# B&R Automation Studio project CamAutomat1
Automation Studio 4.10.5.38 SP; technology packages: mapp 5.23.1, mappCockpit 5.23.0, mappControl 5.23.0, mappMotion 5.23.1, mappView 5.23.0

## Configuration Config1

CPU 5PPC2100.BY44-000, AutomationRuntime A4.83, Build 4.1.2, Safety 0.0, Vc 

CPU 5PPC2200.AL14-000, AutomationRuntime B4.91, Build 4.1.2, Safety 0.0, Vc 

### Task classes (Cpu.sw)
```
Cyclic#1 (cycle 2000 us, tolerance 2000 us):
  CamAutomat <- CamAutomat.prg
  SesnorSim <- SesnorSim.prg
Cyclic#3:
  ComTCP_P <- Libraries.ComTCP.ComTCP_P.prg
Cyclic#4:
  MachineAla <- MachineAlarm.prg
DataObjects: McAcpSys
NcDataObjects: McDriveLog
Binaries: TCData, mvLoader, TCLang, udbdef, arsvcreg, mCoWebSc, arflatprv, arcoal, McAcpDrv, McAcpSim, arconfig, asfw, ashwd, iomap, User, Role, sysconf, TC, ashwac, Config_2, Config, Config_1, Settings, Config_6, TempConfig, Config_7, Config_5, Config_3, Config_4
Libraries: MTBasics, brsystem, MTTypes, sys_lib, runtime, ComTCP_L, operator, astime, AsTCP, standard, AsArLog, AsBrStr, MpRecipe, MpBase, McBase, CoTrace, AsZip, FileIO, MpAxis, McAxis, McAcpAx, MpServer, MpAlarmX, MpCom, MpTemp, asieccon, arssl, asepl, powerlnk, aruser, dataobj
```

### Task classes (Cpu.sw)
```
Cyclic#1 (cycle 2000 us, tolerance 2000 us):
  CamAutomat <- CamAutomat.prg
  TouchProbe <- TouchProbe.prg
Cyclic#4:
  MachineAla <- MachineAlarm.prg
DataObjects: McAcpSys
NcDataObjects: McDriveLog
Binaries: TCData, mvLoader, TCLang, udbdef, arsvcreg, mCoWebSc, arflatprv, arcoal, McAcpDrv, McAcpSim, arconfig, asfw, ashwd, iomap, User, Role, sysconf, TC, ashwac, Config_2, Config, Config_1, Settings, Config_6, TempConfig, Config_5, CamAutom, Config_7, Config_3, Config_4
Libraries: MTBasics, brsystem, MTTypes, sys_lib, runtime, ComTCP_L, operator, astime, AsTCP, standard, AsArLog, AsBrStr, MpRecipe, MpBase, McBase, CoTrace, AsZip, FileIO, MpAxis, McAxis, McAcpAx, MpServer, MpAlarmX, MpCom, MpTemp, asieccon, arssl, asepl, powerlnk, aruser, dataobj
```

### Hardware
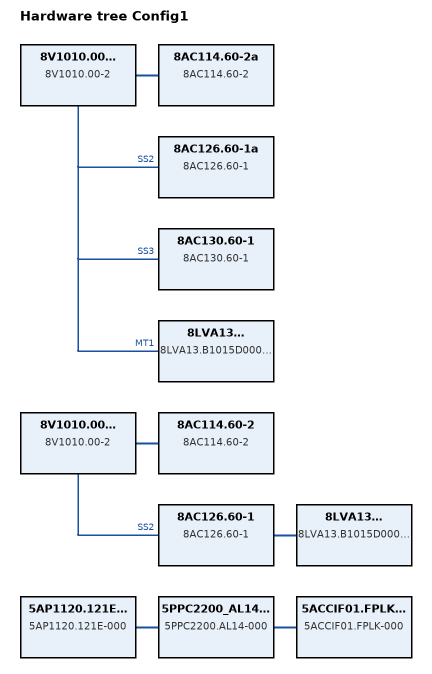
```
5ACCIF01.FPLK-000 : 5ACCIF01.FPLK-000 v1.6.2.0  [SL -> 5PPC2200_AL14_000.SL1]
5AP1120.121E-000 : 5AP1120.121E-000 v2.0.0.0
5PPC2200_AL14_000 : 5PPC2200.AL14-000 v2.0.1.0  [SY -> 5AP1120.121E-000.SY1]
  Connector IF3:
    AssignedOperatingSystem = ARemb
    ActivateDevice = 1
    HostName = mo
    Mode = Manual
    InternetAddress = 192.168.68.70
    SubnetMask = 255.255.255.0
    ActivateSnmp = 2
  Connector IF4:
    AssignedOperatingSystem = GPOS
  Connector IF7:
    OperatingSystem = ARemb
    ActivateDevice = 1
    Mode = Manual
    InternetAddress = 192.168.0.10
    SubnetMask = 255.255.255.0
  Connector IF5:
    AssignedOperatingSystem = ARemb
  Connector IF6:
    AssignedOperatingSystem = GPOS
  ConfigurationID = mappViewGettingStarted_ETA210_T50
  UserPartitionSize = 200
  RemMemDevice = PCI.1.PPC21xx.SRAM
  RemMemSize = 262144
  RemanentGlobalPvSize = 60000
  TimerDeviceType = EPLX2X
  TimerDevice = 5ACCIF01.FPLK-000.IF1
  TaskClassIdleTime = 2000
  Cyclic1Duration = 2000
  Cyclic1Tolerance = 2000
  FileDevice1
  FileDeviceName1 = CSV_Recipes
  FileDevicePath1 = F:\Recipes
  FileDevice2
  FileDeviceName2 = SIM_Recipes
  FileDevicePath2 = C:\Basic
  TimeZone = 65
  FtpUser1
  FtpUsername1 = academy
  FtpUserPassword1 = PTbbKbjlQWNQQLeLnvYxsprPr7USEpMWmZovrSfugvI=
  FtpUserSalt1 = LwThsYzd
  FTPAccessRight1 = 0
  ActivateOpcUa = 1
  OpcUa_SamplingTimer_Selector = 1
  OpcUaInformationModels_PV_Version = 1
  ActivateHypervisor = 1
8AC114.60-2 : 8AC114.60-2 v1.0.0.8  [SS -> 8V1010.00-2Cutter.SS1; PLK1 -> 8AC114.60-2a.PLK1 (NodeNumber=1) [Cable Type=PowerlinkCable, Length=10, Version=1.0.0.3]; PLK2 -> 5ACCIF01.FPLK-000.IF1 (NodeNumber=1) [Cable Type=PowerlinkCable, Length=10, Version=1.0.0.3]]
8AC114.60-2a : 8AC114.60-2 v1.0.0.8  [SS -> 8V1010.00-2aConv.SS1; PLK1 -> 8AC114.60-2.PLK1 (NodeNumber=2) [Cable Type=PowerlinkCable, Length=10, Version=1.0.0.3]]
8AC126.60-1 : 8AC126.60-1 v2.2.0.0  [SS -> 8V1010.00-2Cutter.SS2]
  PlugInType = Encoder
  McAcoposTypeID = AcoposPlugInConfig
8AC126.60-1a : 8AC126.60-1 v2.2.0.0  [SS -> 8V1010.00-2aConv.SS2]
  PlugInType = Encoder
  McAcoposTypeID = AcoposPlugInConfig
8AC130.60-1 : 8AC130.60-1 v2.2.0.0  [SS -> 8V1010.00-2aConv.SS3]
8LVA13.B1015D000-0 : 8LVA13.B1015D000-0 v2.2.0.3  [EC -> 8AC126.60-1.EC; MT -> 8V1010.00-2Cutter.MT1]
  M1/MotorParameters:
    MOTOR_AMB_TEMP_RATED = 40
8LVA13.B1015D000-0a : 8LVA13.B1015D000-0 v2.2.0.3  [MT -> 8V1010.00-2aConv.MT1]
  M1/MotorParameters:
    MOTOR_AMB_TEMP_RATED = 40
8V1010.00-2Cutter : 8V1010.00-2 v2.3.0.0  // Cutter ACOPOS servo drive, 3x 400-480 V, 1.0 A, 0.45 kW, line filter, integrated braking resistor and electronic secure restart inhibit
  DriveConfiguration/Module:
    McAcoposTypeID = AcoposConfig
    ActivateACOPOSSimulationOnPLC = 0
    PowerSupply = ETA
  DriveConfiguration/Channel[1]/RealAxis:
    AxisReference = gCutter_MpLink
    MechanicalElementsIsInvisible = 0
  DriveConfiguration/Channel[1]/RealAxis/MechanicalElements/Gearbox:
    InputIsReadOnly = 0
    Input = 1
    OutputIsReadOnly = 0
    Output = 1
  DriveConfiguration/Channel[1]/RealAxis/MechanicalElements/RotaryToLinearTransformation:
    ReferenceDistanceIsReadOnly = 0
    ReferenceDistance = 360
  DriveConfiguration/Channel[1]/RealAxis/Controller:
    ModeIsReadOnly = 0
    Mode = PositionController
  DriveConfiguration/Channel[1]/RealAxis/Controller/Mode/Position:
    ProportionalGain = 228
    IntegrationTime = 0.0
    PredictionTime = 0.0004
    TotalDelayTime = 0.0004
  DriveConfiguration/Channel[1]/RealAxis/Controller/Mode/Speed:
    ProportionalGainIsReadOnly = 0
    ProportionalGain = 0.599999
    IntegrationTimeIsReadOnly = 0
    IntegrationTime = 0.0
    FilterTimeIsReadOnly = 0
    FilterTime = 0.0
  DriveConfiguration/Channel[1]/RealAxis/Controller/Mode/LoopFilters:
    LoopFilterXIsReadOnly = 0
    LoopFilter1 = NotUsed
    LoopFilter2 = NotUsed
    LoopFilter3 = NotUsed
  DriveConfiguration/Channel[1]/RealAxis/Homing:
    ModeIsReadOnly = 0
    Mode = Direct
  DriveConfiguration/Channel[1]/RealAxis/Homing/Mode:
    Position = 0.0
    ReferencePulse = NotUsed
  DriveConfiguration/Channel[1]/RealAxis/Homing:
    RestorePositionVariable = 
  DriveConfiguration/Channel[1]/RealAxis/StopReaction:
    QuickstopIsReadOnly = 0
    Quickstop = DecelerationLimit
    DriveErrorIsReadOnly = 0
    DriveError = DecelerationLimit
  DriveConfiguration/Channel[1]/RealAxis/MovementErrorLimits:
    PositionError = 1
    VelocityErrorMonitoring = Automatic1
  DriveConfiguration/Channel[1]/RealAxis:
    JerkFilterIsReadOnly = 0
    JerkFilter = NotUsed
    ZeroVibrationFilter = NotUsed
  DriveConfiguration/Channel[1]/RealAxis/DigitalInputs/HomingSwitch:
    SourceIsReadOnly = 0
    Source = X1Ref
    Level = High
  DriveConfiguration/Channel[1]/RealAxis/DigitalInputs/PositiveLimitSwitch:
    Source = X1PosLim
    Level = High
  DriveConfiguration/Channel[1]/RealAxis/DigitalInputs/NegativeLimitSwitch:
    Source = X1NegLim
    Level = High
  DriveConfiguration/Channel[1]/RealAxis/DigitalInputs/Trigger1:
    Source = X1Trigger1
    Level = High
  DriveConfiguration/Channel[1]/RealAxis/DigitalInputs/Trigger2:
    Source = X1Trigger2
    Level = High
  DriveConfiguration/Channel[1]/RealAxis/DigitalInputs/Quickstop:
    Input = NotUsed
  DriveConfiguration/Channel[1]/RealAxis/Simulation:
    SimulationModeOnPLC = SetValueGeneration
    SimulationModeOnACOPOS = NotUsed
  DriveConfiguration/Channel[1]/RealAxis/AxisFeatures:
    FeatureRef[1] = Feature_CamAutomat
  DriveConfiguration/Channel[1]:
    ExternalEncoderAxis = NotUsed
8V1010.00-2aConv : 8V1010.00-2 v2.3.0.0  // Conv ACOPOS servo drive, 3x 400-480 V, 1.0 A, 0.45 kW, line filter, integrated braking resistor and electronic secure restart inhibit
  DriveConfiguration/Module:
    McAcoposTypeID = AcoposConfig
    ActivateACOPOSSimulationOnPLC = 0
    PowerSupply = ETA
  DriveConfiguration/Channel[1]/RealAxis:
    AxisReference = gConv_MpLink
    MechanicalElementsIsInvisible = 0
  DriveConfiguration/Channel[1]/RealAxis/MechanicalElements/Gearbox:
    InputIsReadOnly = 0
    Input = 1
    OutputIsReadOnly = 0
    Output = 1
  DriveConfiguration/Channel[1]/RealAxis/MechanicalElements/RotaryToLinearTransformation:
    ReferenceDistanceIsReadOnly = 0
    ReferenceDistance = 160
  DriveConfiguration/Channel[1]/RealAxis/Controller:
    ModeIsReadOnly = 0
    Mode = PositionController
  DriveConfiguration/Channel[1]/RealAxis/Controller/Mode/Position:
    ProportionalGain = 269
    IntegrationTime = 0.0
    PredictionTime = 0.0004
    TotalDelayTime = 0.0004
  DriveConfiguration/Channel[1]/RealAxis/Controller/Mode/Speed:
    ProportionalGainIsReadOnly = 0
    ProportionalGain = 0.45
    IntegrationTimeIsReadOnly = 0
    IntegrationTime = 0.0
    FilterTimeIsReadOnly = 0
    FilterTime = 0.0
  DriveConfiguration/Channel[1]/RealAxis/Controller/Mode/LoopFilters:
    LoopFilterXIsReadOnly = 0
    LoopFilter1 = NotUsed
    LoopFilter2 = NotUsed
    LoopFilter3 = NotUsed
  DriveConfiguration/Channel[1]/RealAxis/Homing:
    ModeIsReadOnly = 0
    Mode = Direct
  DriveConfiguration/Channel[1]/RealAxis/Homing/Mode:
    Position = 0.0
    ReferencePulse = NotUsed
  DriveConfiguration/Channel[1]/RealAxis/Homing:
    RestorePositionVariable = 
  DriveConfiguration/Channel[1]/RealAxis/StopReaction:
    QuickstopIsReadOnly = 0
    Quickstop = DecelerationLimit
    DriveErrorIsReadOnly = 0
    DriveError = DecelerationLimit
  DriveConfiguration/Channel[1]/RealAxis/MovementErrorLimits:
    PositionError = 1
    VelocityErrorMonitoring = Automatic1
  DriveConfiguration/Channel[1]/RealAxis:
    JerkFilterIsReadOnly = 0
    JerkFilter = NotUsed
    ZeroVibrationFilter = NotUsed
  DriveConfiguration/Channel[1]/RealAxis/DigitalInputs/HomingSwitch:
    SourceIsReadOnly = 0
    Source = X1Ref
    Level = High
  DriveConfiguration/Channel[1]/RealAxis/DigitalInputs/PositiveLimitSwitch:
    Source = X1PosLim
    Level = High
  DriveConfiguration/Channel[1]/RealAxis/DigitalInputs/NegativeLimitSwitch:
    Source = X1NegLim
    Level = High
  DriveConfiguration/Channel[1]/RealAxis/DigitalInputs/Trigger1:
    Source = X1Trigger1
    Level = High
  DriveConfiguration/Channel[1]/RealAxis/DigitalInputs/Trigger2:
    Source = X1Trigger2
    Level = High
  DriveConfiguration/Channel[1]/RealAxis/DigitalInputs/Quickstop:
    Input = NotUsed
  DriveConfiguration/Channel[1]/RealAxis/Simulation:
    SimulationModeOnPLC = SetValueGeneration
    SimulationModeOnACOPOS = NotUsed
  DriveConfiguration/Channel[1]/RealAxis/AxisFeatures:
    FeatureRef[1] = 
  DriveConfiguration/Channel[1]:
    ExternalEncoderAxis = NotUsed
```

### TempConfig.tempcontroller - 5PPC2100_BY44_000/mappControl/TempConfig.tempcontroller
```
Element gTempController_2 (Type=tempcontroller)
  TempController:
    SoftStart = NotUsed
Element gTempController_1 (Type=tempcontroller)
  TempController:
    SoftStart = NotUsed
```

### CamAutom.axisfeature - 5PPC2100_BY44_000/mappMotion/CamAutom.axisfeature
```
Element Feature_CamAutomat_1 (Type=axisfeature)
  Type = CamAutomat
    CamAutomatType = ACOPOS
      CommonParameters:
        Master:
          ValueSource = SetPosition
            AxisReference = gAxis1_MpLink
            MaxVelocity = 1000
          StartPosition = 0.0
          StartInterval = MasterAxisPeriod
        AdvancedParameters:
          StartStateParameters:
            StartState = 0
            RelMasterStartPos = 0.0
          AdditiveAxes:
            AdditiveMasterValueSource = NotUsed
            AdditiveSlaveValueSource = NotUsed
          MasterStartPositionMode = NotEvaluatedAnew
          ControlSettings:
            CrossLeftBoundary = PositionLimitedHorizontal
            CamChangeImmediately = CurrentMasterMoveDir
          MessageSettings:
            ErrorsInStandby = NoErrorMessages
          TriggerAndLatch:
            Trigger1Delay = 0.0
            Trigger2Delay = 0.0
            SlaveLatchParID = 0
          EventParIDs
          StartIntervals
          Factors:
            SlaveFactorParID = 0
      States:
        State0 = Used
          Events:
            Event[0]:
              Type = MasterStartPosition
              Transition = Immediately
              SynchronousUpdate = NotUsed
              NextState = 1
        State[1]:
          Cam = Predefined
            PredefinedCam = OneToOne
          MasterFactor = 72
          SlaveFactor = 0
          CompensationMode = DistancesBetweenCamCenterPoints
            MasterDistance = 288
            SlaveDistance = 0.0
            AdvancedParameters = NotUsed
          AdvancedParameters:
            RepeatCounterInit = 0
            MasterValueSource = CommonMaster
          Events:
            Event[0]:
              Type = Signal1FromPLC
              Transition = EndOfState
              SynchronousUpdate = NotUsed
              NextState = 2
        State[2]:
          Cam = Predefined
            PredefinedCam = OneToOne
          MasterFactor = 72
          SlaveFactor = 72
          CompensationMode = MaDistBetweenLatchPosCenter
            MasterDistance = 144
            SlaveDistance = 144
            AdvancedParameters = NotUsed
          AdvancedParameters:
            RepeatCounterInit = 0
            MasterValueSource = CommonMaster
          Events:
            Event[0]:
              Type = Signal1FromPLC
              Transition = EndOfState
              SynchronousUpdate = NotUsed
              NextState = 3
            Event[1]:
              Type = StateEnd
              Transition = EndOfState
              SynchronousUpdate = NotUsed
              NextState = 4
        State[3]:
          Cam = Predefined
            PredefinedCam = OneToOne
          MasterFactor = 72
          SlaveFactor = 72
          CompensationMode = MaDistBetweenLatchPosCenter
            MasterDistance = 288
            SlaveDistance = 288
            AdvancedParameters = NotUsed
          AdvancedParameters:
            RepeatCounterInit = 0
            MasterValueSource = CommonMaster
          Events:
            Event[0]:
              Type = Signal1FromPLC
              Transition = EndOfState
              SynchronousUpdate = NotUsed
              NextState = 3
            Event[1]:
              Type = StateEnd
              Transition = EndOfState
              SynchronousUpdate = NotUsed
              NextState = 4
        State[4]:
          Cam = Predefined
            PredefinedCam = OneToOne
          MasterFactor = 72
          SlaveFactor = 0
          CompensationMode = MaDistBetweenLatchPosCenter
            MasterDistance = 144
            SlaveDistance = 144
            AdvancedParameters = NotUsed
          AdvancedParameters:
            RepeatCounterInit = 0
            MasterValueSource = CommonMaster
          Events:
            Event[0]:
              Type = Signal1FromPLC
              Transition = EndOfState
              SynchronousUpdate = NotUsed
              NextState = 2
            Event[1]:
              Type = StateEnd
              Transition = EndOfState
              SynchronousUpdate = NotUsed
              NextState = 1
Element Feature_CamAutomat (Type=axisfeature)
  Type = CamAutomat
    CamAutomatType = ACOPOS
      CommonParameters:
        Master:
          ValueSource = SetPosition
            AxisReference = gAxis1_MpLink
            MaxVelocity = 1000
          StartPosition = 0.0
          StartInterval = MasterAxisPeriod
        AdvancedParameters:
          StartStateParameters:
            StartState = 0
            RelMasterStartPos = 0.0
          AdditiveAxes:
            AdditiveMasterValueSource = NotUsed
            AdditiveSlaveValueSource = NotUsed
          MasterStartPositionMode = NotEvaluatedAnew
          ControlSettings:
            CrossLeftBoundary = PositionLimitedHorizontal
            CamChangeImmediately = CurrentMasterMoveDir
          MessageSettings:
            ErrorsInStandby = NoErrorMessages
          TriggerAndLatch:
            Trigger1Delay = 0.0
            Trigger2Delay = 0.0
            SlaveLatchParID = 0
          EventParIDs
          StartIntervals
          Factors:
            SlaveFactorParID = 0
      States:
        State0 = Used
          Events:
            Event[0]:
              Type = MasterStartPosition
              Transition = Immediately
              SynchronousUpdate = NotUsed
              NextState = 1
        State[1]:
          Cam = Predefined
            PredefinedCam = OneToOne
          MasterFactor = 1
          SlaveFactor = 0
          CompensationMode = DistancesBetweenCamCenterPoints
            MasterDistance = 0.0
            SlaveDistance = 0.0
            AdvancedParameters = NotUsed
          AdvancedParameters:
            RepeatCounterInit = 0
            MasterValueSource = CommonMaster
          Events:
            Event[0]:
              Type = Signal1FromPLC
              Transition = EndOfState
              SynchronousUpdate = NotUsed
              NextState = 2
        State[2]:
          Cam = Predefined
            PredefinedCam = OneToOne
          MasterFactor = 1
          SlaveFactor = 1
          CompensationMode = MaDistBetweenLatchPosCenter
            MasterDistance = 130
            SlaveDistance = 170
            AdvancedParameters = NotUsed
          AdvancedParameters:
            RepeatCounterInit = 0
            MasterValueSource = CommonMaster
          Events:
            Event[0]:
              Type = StateEnd
              Transition = EndOfState
              SynchronousUpdate = NotUsed
              NextState = 3
        State[3]:
          Cam = Predefined
            PredefinedCam = OneToOne
          MasterFactor = 1
          SlaveFactor = 1
          CompensationMode = MaDistBetweenLatchPosCenter
            MasterDistance = 20
            SlaveDistance = 20
            AdvancedParameters = NotUsed
          AdvancedParameters:
            RepeatCounterInit = 0
            MasterValueSource = CommonMaster
          Events:
            Event[0]:
              Type = StateEnd
              Transition = EndOfState
              SynchronousUpdate = NotUsed
              NextState = 4
        State[4]:
          Cam = Predefined
            PredefinedCam = OneToOne
          MasterFactor = 1
          SlaveFactor = 0
          CompensationMode = MaDistBetweenLatchPosCenter
            MasterDistance = 130
            SlaveDistance = 170
            AdvancedParameters = NotUsed
          AdvancedParameters:
            RepeatCounterInit = 0
            MasterValueSource = CommonMaster
          Events:
            Event[0]:
              Type = StateEnd
              Transition = EndOfState
              SynchronousUpdate = NotUsed
              NextState = 1
```

### Config_1.axis - 5PPC2100_BY44_000/mappMotion/Config_1.axis
```
Element gAxis2_MpLink (Type=axis)
  BaseTypeIsReadOnly = 0
  BaseType = RotaryPeriodic
    MeasurementUnitIsReadOnly = 0
    MeasurementUnit = 17476
    MeasurementResolutionIsReadOnly = 0
    MeasurementResolution = 1
    CountDirectionIsReadOnly = 0
    CountDirection = Standard
    PeriodSettings:
      Period = 360.0
  MovementLimitsIsReadOnly = 0
  MovementLimits = Internal
    Position:
      LowerLimitMin = -1.79769313486231E308
      UpperLimitMax = 1.79769313486231E308
      LowerLimit = -1000.0
      UpperLimit = 1000.0
    VelocityIsReadOnly = 0
    Velocity:
      VelocityMax = 3.4E38
      Velocity = 6000
    AccelerationIsReadOnly = 0
    Acceleration:
      AccelerationMax = 3.4E38
      Acceleration = 60000
    DecelerationIsReadOnly = 0
    Deceleration:
      DecelerationMax = 3.4E38
      Deceleration = 60000
  Alarms = MpAlarmX
Element gAxis1_MpLink (Type=axis)
  BaseTypeIsReadOnly = 0
  BaseType = RotaryPeriodic
    MeasurementUnitIsReadOnly = 0
    MeasurementUnit = 17476
    MeasurementResolutionIsReadOnly = 0
    MeasurementResolution = 1
    CountDirectionIsReadOnly = 0
    CountDirection = Standard
    PeriodSettings:
      Period = 360.0
  MovementLimitsIsReadOnly = 0
  MovementLimits = Internal
    Position:
      LowerLimitMin = -1.79769313486231E308
      UpperLimitMax = 1.79769313486231E308
      LowerLimit = -1000.0
      UpperLimit = 1000.0
    VelocityIsReadOnly = 0
    Velocity:
      VelocityMax = 3.4E38
      Velocity = 6000
    AccelerationIsReadOnly = 0
    Acceleration:
      AccelerationMax = 3.4E38
      Acceleration = 60000
    DecelerationIsReadOnly = 0
    Deceleration:
      DecelerationMax = 3.4E38
      Deceleration = 60000
  Alarms = MpAlarmX
```

### Axis.axis - 5PPC2200_AL14_000/mappMotion/Axis.axis
```
Element gConv_MpLink (Type=axis)  // Conver Servo
  BaseTypeIsReadOnly = 0
  BaseType = LinearPeriodic
    MeasurementUnit = 5066068
    MeasurementResolutionIsReadOnly = 0
    MeasurementResolution = 0.01
    CountDirectionIsReadOnly = 0
    CountDirection = Standard
    PeriodSettings:
      Period = 144
  MovementLimitsIsReadOnly = 0
  MovementLimits = Internal
    Position:
      LowerLimitMin = -1.79769313486231E308
      UpperLimitMax = 1.79769313486231E308
      LowerLimit = -1000.0
      UpperLimit = 1000.0
    VelocityIsReadOnly = 0
    Velocity:
      VelocityMax = 3.4E38
      Velocity = 6000
    AccelerationIsReadOnly = 0
    Acceleration:
      AccelerationMax = 3.4E38
      Acceleration = 60000
    DecelerationIsReadOnly = 0
    Deceleration:
      DecelerationMax = 3.4E38
      Deceleration = 60000
  Alarms = MpAlarmX
Element gCutter_MpLink (Type=axis)  // Cutter Servo
  BaseTypeIsReadOnly = 0
  BaseType = RotaryPeriodic
    MeasurementUnitIsReadOnly = 0
    MeasurementUnit = 17476
    MeasurementResolutionIsReadOnly = 0
    MeasurementResolution = 0.01
    CountDirectionIsReadOnly = 0
    CountDirection = Inverse
    PeriodSettings:
      Period = 360
  MovementLimitsIsReadOnly = 0
  MovementLimits = Internal
    Position:
      LowerLimitMin = -1.79769313486231E308
      UpperLimitMax = 1.79769313486231E308
      LowerLimit = -1000.0
      UpperLimit = 1000.0
    VelocityIsReadOnly = 0
    Velocity:
      VelocityMax = 3.4E38
      Velocity = 6000
    AccelerationIsReadOnly = 0
    Acceleration:
      AccelerationMax = 3.4E38
      Acceleration = 60000
    DecelerationIsReadOnly = 0
    Deceleration:
      DecelerationMax = 3.4E38
      Deceleration = 60000
  Alarms = MpAlarmX
```

### CamAutom.axisfeature - 5PPC2200_AL14_000/mappMotion/CamAutom.axisfeature
```
Element Feature_CamAutomatbak (Type=axisfeature)
  Type = CamAutomat
    CamAutomatType = ACOPOS
      CommonParameters:
        Master:
          ValueSource = SetPosition
            AxisReference = gConv_MpLink
            MaxVelocity = 1000
          StartPosition = 0.00
          StartInterval = MasterAxisPeriod
        AdvancedParameters:
          StartStateParameters:
            StartState = 0
            RelMasterStartPos = 0.0
          AdditiveAxes:
            AdditiveMasterValueSource = NotUsed
            AdditiveSlaveValueSource = NotUsed
          MasterStartPositionMode = NotEvaluatedAnew
          ControlSettings:
            CrossLeftBoundary = PositionLimitedHorizontal
            CamChangeImmediately = CurrentMasterMoveDir
          MessageSettings:
            ErrorsInStandby = NoErrorMessages
          TriggerAndLatch:
            Trigger1Delay = 0.0
            Trigger2Delay = 0.0
            SlaveLatchParID = 0
          EventParIDs
          StartIntervals
          Factors:
            SlaveFactorParID = 0
      States:
        State0 = Used
          Events:
            Event[0]:
              Type = MasterStartPosition
              Transition = Immediately
              SynchronousUpdate = NotUsed
              NextState = 1
        State[1]:
          Cam = Predefined
            PredefinedCam = OneToOne
          MasterFactor = 100
          SlaveFactor = 0
          CompensationMode = DistancesBetweenExitEntryPoints
            MasterDistance = 0
            SlaveDistance = 0
            AdvancedParameters = NotUsed
          AdvancedParameters:
            RepeatCounterInit = 0
            MasterValueSource = CommonMaster
          Events:
            Event[0]:
              Type = Signal1FromPLC
              Transition = EndOfState
              SynchronousUpdate = NotUsed
              NextState = 2
        State[2]:
          Cam = Predefined
            PredefinedCam = OneToOne
          MasterFactor = 2000
          SlaveFactor = 2300
          CompensationMode = DistancesBetweenExitEntryPoints
            MasterDistance = 100
            SlaveDistance = 160
            AdvancedParameters = NotUsed
          AdvancedParameters:
            RepeatCounterInit = 0
            MasterValueSource = CommonMaster
          Events:
            Event[0]:
              Type = StateEnd
              Transition = EndOfState
              SynchronousUpdate = NotUsed
              NextState = 3
        State[3]:
          Cam = Predefined
            PredefinedCam = OneToOne
          MasterFactor = 100
          SlaveFactor = 0
          CompensationMode = DistancesBetweenExitEntryPoints
            MasterDistance = 1
            SlaveDistance = 288
            AdvancedParameters = NotUsed
          AdvancedParameters:
            RepeatCounterInit = 0
            MasterValueSource = CommonMaster
          Events:
            Event[0]:
              Type = Signal1FromPLC
              Transition = EndOfState
              SynchronousUpdate = NotUsed
              NextState = 3
            Event[1]:
              Type = StateEnd
              Transition = Immediately
              SynchronousUpdate = NotUsed
              NextState = 4
        State[4]:
          Cam = Predefined
            PredefinedCam = OneToOne
          MasterFactor = 72
          SlaveFactor = 0
          CompensationMode = DistancesBetweenExitEntryPoints
            MasterDistance = 144
            SlaveDistance = 144
            AdvancedParameters = NotUsed
          AdvancedParameters:
            RepeatCounterInit = 0
            MasterValueSource = CommonMaster
          Events:
            Event[0]:
              Type = Signal1FromPLC
              Transition = EndOfState
              SynchronousUpdate = NotUsed
              NextState = 2
            Event[1]:
              Type = StateEnd
              Transition = Immediately
              SynchronousUpdate = NotUsed
              NextState = 1
Element Feature_CamAutomat_3rd (Type=axisfeature)
  Type = CamAutomat
    CamAutomatType = ACOPOS
      CommonParameters:
        Master:
          ValueSource = SetPosition
            AxisReference = gConv_MpLink
            MaxVelocity = 1000
          StartPosition = 0.00
          StartInterval = MasterAxisPeriod
        AdvancedParameters:
          StartStateParameters:
            StartState = 0
            RelMasterStartPos = 0.0
          AdditiveAxes:
            AdditiveMasterValueSource = NotUsed
            AdditiveSlaveValueSource = NotUsed
          MasterStartPositionMode = NotEvaluatedAnew
          ControlSettings:
            CrossLeftBoundary = PositionLimitedHorizontal
            CamChangeImmediately = CurrentMasterMoveDir
          MessageSettings:
            ErrorsInStandby = NoErrorMessages
          TriggerAndLatch:
            Trigger1Delay = 0.0
            Trigger2Delay = 0.0
            SlaveLatchParID = 0
          EventParIDs
          StartIntervals
          Factors:
            SlaveFactorParID = 0
      States:
        State0 = Used
          Events:
            Event[0]:
              Type = MasterStartPosition
              Transition = Immediately
              SynchronousUpdate = NotUsed
              NextState = 1
        State[1]:
          Cam = Predefined
            PredefinedCam = OneToOne
          MasterFactor = 100
          SlaveFactor = 0
          CompensationMode = NoCompensation
          AdvancedParameters:
            RepeatCounterInit = 0
            MasterValueSource = CommonMaster
          Events:
            Event[0]:
              Type = Signal1FromPLC
              Transition = EndOfState
              SynchronousUpdate = NotUsed
              NextState = 2
        State[2]:
          Cam = Predefined
            PredefinedCam = OneToOne
          MasterFactor = 2000
          SlaveFactor = 2000
          CompensationMode = DistancesBetweenExitEntryPoints
            MasterDistance = 95
            SlaveDistance = 80
            AdvancedParameters = NotUsed
          AdvancedParameters:
            RepeatCounterInit = 0
            MasterValueSource = CommonMaster
          Events:
            Event[0]:
              Type = Signal1FromPLC
              Transition = EndOfState
              SynchronousUpdate = NotUsed
              NextState = 4
            Event[1]:
              Type = StateEnd
              Transition = EndOfState
              SynchronousUpdate = NotUsed
              NextState = 3
        State[3]:
          Cam = Predefined
            PredefinedCam = OneToOne
          MasterFactor = 100
          SlaveFactor = 0
          CompensationMode = NoCompensation
          AdvancedParameters:
            RepeatCounterInit = 0
            MasterValueSource = CommonMaster
          Events:
            Event[0]:
              Type = Signal1FromPLC
              Transition = EndOfState
              SynchronousUpdate = NotUsed
              NextState = 4
            Event[1]:
              Type = Signal2FromPLC
              Transition = Immediately
              SynchronousUpdate = NotUsed
              NextState = 5
        State[4]:
          Cam = Predefined
            PredefinedCam = OneToOne
          MasterFactor = 2000
          SlaveFactor = 2000
          CompensationMode = DistancesBetweenExitEntryPoints
            MasterDistance = 50
            SlaveDistance = 340
            AdvancedParameters = NotUsed
          AdvancedParameters:
            RepeatCounterInit = 0
            MasterValueSource = CommonMaster
          Events:
            Event[0]:
              Type = StateEnd
              Transition = Immediately
              SynchronousUpdate = NotUsed
              NextState = 3
        State[5]:
          Cam = Predefined
            PredefinedCam = OneToOne
          MasterFactor = 100
          SlaveFactor = 0
          CompensationMode = DistancesBetweenExitEntryPoints
            MasterDistance = 260
            SlaveDistance = 260
            AdvancedParameters = NotUsed
          AdvancedParameters:
            RepeatCounterInit = 0
            MasterValueSource = CommonMaster
          Events:
            Event[0]:
              Type = StateEnd
              Transition = EndOfState
              SynchronousUpdate = NotUsed
              NextState = 6
        State[6]:
          Cam = Predefined
            PredefinedCam = OneToOne
          MasterFactor = 100
          SlaveFactor = 0
          CompensationMode = NoCompensation
          AdvancedParameters:
            RepeatCounterInit = 0
            MasterValueSource = CommonMaster
Element Feature_CamAutomat_2nd (Type=axisfeature)
  Type = CamAutomat
    CamAutomatType = ACOPOS
      CommonParameters:
        Master:
          ValueSource = SetPosition
            AxisReference = gConv_MpLink
            MaxVelocity = 1000
          StartPosition = 0.00
          StartInterval = MasterAxisPeriod
        AdvancedParameters:
          StartStateParameters:
            StartState = 0
            RelMasterStartPos = 0.0
          AdditiveAxes:
            AdditiveMasterValueSource = NotUsed
            AdditiveSlaveValueSource = NotUsed
          MasterStartPositionMode = NotEvaluatedAnew
          ControlSettings:
            CrossLeftBoundary = PositionLimitedHorizontal
            CamChangeImmediately = CurrentMasterMoveDir
          MessageSettings:
            ErrorsInStandby = NoErrorMessages
          TriggerAndLatch:
            Trigger1Delay = 0.0
            Trigger2Delay = 0.0
            SlaveLatchParID = 0
          EventParIDs
          StartIntervals
          Factors:
            SlaveFactorParID = 0
      States:
        State0 = Used
          Events:
            Event[0]:
              Type = MasterStartPosition
              Transition = Immediately
              SynchronousUpdate = NotUsed
              NextState = 1
        State[1]:
          Cam = Predefined
            PredefinedCam = OneToOne
          MasterFactor = 100
          SlaveFactor = 0
          CompensationMode = NoCompensation
          AdvancedParameters:
            RepeatCounterInit = 0
            MasterValueSource = CommonMaster
          Events:
            Event[0]:
              Type = Signal1FromPLC
              Transition = EndOfState
              SynchronousUpdate = NotUsed
              NextState = 2
        State[2]:
          Cam = Predefined
            PredefinedCam = OneToOne
          MasterFactor = 2000
          SlaveFactor = 2000
          CompensationMode = DistancesBetweenExitEntryPoints
            MasterDistance = 95
            SlaveDistance = 160
            AdvancedParameters = NotUsed
          AdvancedParameters:
            RepeatCounterInit = 0
            MasterValueSource = CommonMaster
          Events:
            Event[0]:
              Type = Signal1FromPLC
              Transition = EndOfState
              SynchronousUpdate = NotUsed
              NextState = 4
            Event[1]:
              Type = StateEnd
              Transition = EndOfState
              SynchronousUpdate = NotUsed
              NextState = 3
        State[3]:
          Cam = Predefined
            PredefinedCam = OneToOne
          MasterFactor = 1000
          SlaveFactor = 1000
          CompensationMode = DistancesBetweenExitEntryPoints
            MasterDistance = 20
            SlaveDistance = 170
            AdvancedParameters = NotUsed
          AdvancedParameters:
            RepeatCounterInit = 0
            MasterValueSource = CommonMaster
          Events:
            Event[0]:
              Type = Signal1FromPLC
              Transition = EndOfState
              SynchronousUpdate = NotUsed
              NextState = 6
        State[4]:
          Cam = Predefined
            PredefinedCam = OneToOne
          MasterFactor = 2000
          SlaveFactor = 2000
          CompensationMode = DistancesBetweenExitEntryPoints
            MasterDistance = 95
            SlaveDistance = 340
            AdvancedParameters = NotUsed
          AdvancedParameters:
            RepeatCounterInit = 0
            MasterValueSource = CommonMaster
          Events:
            Event[0]:
              Type = Signal1FromPLC
              Transition = EndOfState
              SynchronousUpdate = NotUsed
              NextState = 5
            Event[1]:
              Type = StateEnd
              Transition = Immediately
              SynchronousUpdate = NotUsed
              NextState = 3
        State[5]:
          Cam = Predefined
            PredefinedCam = OneToOne
          MasterFactor = 2000
          SlaveFactor = 2000
          CompensationMode = DistancesBetweenExitEntryPoints
            MasterDistance = 95
            SlaveDistance = 340
            AdvancedParameters = NotUsed
          AdvancedParameters:
            RepeatCounterInit = 0
            MasterValueSource = CommonMaster
          Events:
            Event[0]:
              Type = Signal1FromPLC
              Transition = EndOfState
              SynchronousUpdate = NotUsed
              NextState = 4
            Event[1]:
              Type = StateEnd
              Transition = EndOfState
              SynchronousUpdate = NotUsed
              NextState = 3
        State[6]:
          Cam = Predefined
            PredefinedCam = OneToOne
          MasterFactor = 2000
          SlaveFactor = 2000
          CompensationMode = DistancesBetweenExitEntryPoints
            MasterDistance = 25
            SlaveDistance = 160
            AdvancedParameters = NotUsed
          AdvancedParameters:
            RepeatCounterInit = 0
            MasterValueSource = CommonMaster
          Events:
            Event[0]:
              Type = Signal1FromPLC
              Transition = EndOfState
              SynchronousUpdate = NotUsed
              NextState = 5
            Event[1]:
              Type = StateEnd
              Transition = EndOfState
              SynchronousUpdate = NotUsed
              NextState = 3
Element Feature_CamAutomat_finalok (Type=axisfeature)
  Type = CamAutomat
    CamAutomatType = ACOPOS
      CommonParameters:
        Master:
          ValueSource = SetPosition
            AxisReference = gConv_MpLink
            MaxVelocity = 1000
          StartPosition = 0.00
          StartInterval = SpecifyValue
            Interval = 1.0
        AdvancedParameters:
          StartStateParameters:
            StartState = 0
            RelMasterStartPos = 0.0
          AdditiveAxes:
            AdditiveMasterValueSource = NotUsed
            AdditiveSlaveValueSource = NotUsed
          MasterStartPositionMode = NotEvaluatedAnew
          ControlSettings:
            CrossLeftBoundary = PositionLimitedHorizontal
            CamChangeImmediately = CurrentMasterMoveDir
          MessageSettings:
            ErrorsInStandby = NoErrorMessages
          TriggerAndLatch:
            Trigger1Delay = 0.0
            Trigger2Delay = 0.0
            SlaveLatchParID = 0
          EventParIDs
          StartIntervals
          Factors:
            SlaveFactorParID = 0
      States:
        State0 = Used
          Events:
            Event[0]:
              Type = MasterStartPosition
              Transition = Immediately
              SynchronousUpdate = NotUsed
              NextState = 1
        State[1]:
          Cam = Predefined
            PredefinedCam = OneToOne
          MasterFactor = 100
          SlaveFactor = 0
          CompensationMode = NoCompensation
          AdvancedParameters:
            RepeatCounterInit = 0
            MasterValueSource = CommonMaster
          Events:
            Event[0]:
              Type = Signal1FromPLC
              Transition = EndOfState
              SynchronousUpdate = NotUsed
              NextState = 2
        State[2]:
          Cam = Predefined
            PredefinedCam = OneToOne
          MasterFactor = 100
          SlaveFactor = 0
          CompensationMode = DistancesBetweenExitEntryPoints
            MasterDistance = 27
            SlaveDistance = 80
            AdvancedParameters = NotUsed
          AdvancedParameters:
            RepeatCounterInit = 0
            MasterValueSource = CommonMaster
          Events:
            Event[0]:
              Type = StateEnd
              Transition = EndOfState
              SynchronousUpdate = NotUsed
              NextState = 3
        State[3]:
          Cam = Predefined
            PredefinedCam = OneToOne
          MasterFactor = 2000
          SlaveFactor = 2000
          CompensationMode = DistancesBetweenExitEntryPoints
            MasterDistance = 0
            SlaveDistance = 0
            AdvancedParameters = NotUsed
          AdvancedParameters:
            RepeatCounterInit = 0
            MasterValueSource = CommonMaster
          Events:
            Event[0]:
              Type = StateEnd
              Transition = EndOfState
              SynchronousUpdate = NotUsed
              NextState = 4
        State[4]:
          Cam = Predefined
            PredefinedCam = OneToOne
          MasterFactor = 100
          SlaveFactor = 1
          CompensationMode = DistancesBetweenExitEntryPoints
            MasterDistance = 16
            SlaveDistance = 260
            AdvancedParameters = NotUsed
          AdvancedParameters:
            RepeatCounterInit = 0
            MasterValueSource = CommonMaster
          Events:
            Event[0]:
              Type = StateEnd
              Transition = EndOfState
              SynchronousUpdate = NotUsed
              NextState = 1
Element Feature_CamAutomat (Type=axisfeature)
  Type = CamAutomat
    CamAutomatType = ACOPOS
      CommonParameters:
        Master:
          ValueSource = SetPosition
            AxisReference = gConv_MpLink
            MaxVelocity = 1000
          StartPosition = 0.00
          StartInterval = SpecifyValue
            Interval = 1.0
        AdvancedParameters:
          StartStateParameters:
            StartState = 0
            RelMasterStartPos = 0.0
          AdditiveAxes:
            AdditiveMasterValueSource = NotUsed
            AdditiveSlaveValueSource = NotUsed
          MasterStartPositionMode = NotEvaluatedAnew
          ControlSettings:
            CrossLeftBoundary = PositionLimitedHorizontal
            CamChangeImmediately = CurrentMasterMoveDir
          MessageSettings:
            ErrorsInStandby = NoErrorMessages
          TriggerAndLatch:
            Trigger1Delay = 0.0
            Trigger2Delay = 0.0
            SlaveLatchParID = 0
          EventParIDs
          StartIntervals
          Factors:
            SlaveFactorParID = 0
      States:
        State0 = Used
          Events:
            Event[0]:
              Type = MasterStartPosition
              Transition = Immediately
              SynchronousUpdate = NotUsed
              NextState = 1
        State[1]:
          Cam = Predefined
            PredefinedCam = OneToOne
          MasterFactor = 100
          SlaveFactor = 0
          CompensationMode = NoCompensation
          AdvancedParameters:
            RepeatCounterInit = 0
            MasterValueSource = CommonMaster
          Events:
            Event[0]:
              Type = Signal1FromPLC
              Transition = EndOfState
              SynchronousUpdate = NotUsed
              NextState = 2
            Event[1]:
              Type = Signal2FromPLC
              Transition = EndOfState
              SynchronousUpdate = NotUsed
              NextState = 5
        State[2]:
          Cam = Predefined
            PredefinedCam = OneToOne
          MasterFactor = 100
          SlaveFactor = 0
          CompensationMode = DistancesBetweenExitEntryPoints
            MasterDistance = 27
            SlaveDistance = 82
            AdvancedParameters = NotUsed
          AdvancedParameters:
            RepeatCounterInit = 0
            MasterValueSource = CommonMaster
          Events:
            Event[0]:
              Type = StateEnd
              Transition = EndOfState
              SynchronousUpdate = NotUsed
              NextState = 3
        State[3]:
          Cam = Predefined
            PredefinedCam = OneToOne
          MasterFactor = 2000
          SlaveFactor = 2200
          CompensationMode = DistancesBetweenExitEntryPoints
            MasterDistance = 0
            SlaveDistance = 0
            AdvancedParameters = NotUsed
          AdvancedParameters:
            RepeatCounterInit = 0
            MasterValueSource = CommonMaster
          Events:
            Event[0]:
              Type = StateEnd
              Transition = EndOfState
              SynchronousUpdate = NotUsed
              NextState = 4
        State[4]:
          Cam = Predefined
            PredefinedCam = OneToOne
          MasterFactor = 100
          SlaveFactor = 0
          CompensationMode = DistancesBetweenExitEntryPoints
            MasterDistance = 16
            SlaveDistance = 256
            AdvancedParameters = NotUsed
          AdvancedParameters:
            RepeatCounterInit = 0
            MasterValueSource = CommonMaster
          Events:
            Event[0]:
              Type = StateEnd
              Transition = EndOfState
              SynchronousUpdate = NotUsed
              NextState = 1
        State[5]:
          Cam = Predefined
            PredefinedCam = OneToOne
          MasterFactor = 100
          SlaveFactor = 0
          CompensationMode = DistancesBetweenExitEntryPoints
            MasterDistance = 27
            SlaveDistance = 82
            AdvancedParameters = NotUsed
          AdvancedParameters:
            RepeatCounterInit = 0
            MasterValueSource = CommonMaster
          Events:
            Event[0]:
              Type = StateEnd
              Transition = EndOfState
              SynchronousUpdate = NotUsed
              NextState = 6
        State[6]:
          Cam = Predefined
            PredefinedCam = OneToOne
          MasterFactor = 2000
          SlaveFactor = 2200
          CompensationMode = DistancesBetweenExitEntryPoints
            MasterDistance = 0
            SlaveDistance = 0
            AdvancedParameters = NotUsed
          AdvancedParameters:
            RepeatCounterInit = 0
            MasterValueSource = CommonMaster
          Events:
            Event[0]:
              Type = StateEnd
              Transition = EndOfState
              SynchronousUpdate = NotUsed
              NextState = 7
        State[7]:
          Cam = Predefined
            PredefinedCam = OneToOne
          MasterFactor = 100
          SlaveFactor = 0
          CompensationMode = DistancesBetweenExitEntryPoints
            MasterDistance = 16
            SlaveDistance = 76
            AdvancedParameters = NotUsed
          AdvancedParameters:
            RepeatCounterInit = 0
            MasterValueSource = CommonMaster
          Events:
            Event[0]:
              Type = StateEnd
              Transition = EndOfState
              SynchronousUpdate = NotUsed
              NextState = 1
```

### Config_1.axis - 5PPC2200_AL14_000/mappMotion/Config_1.axis
```
Element gConv_MpLink (Type=axis)
  BaseTypeIsReadOnly = 0
  BaseType = LinearPeriodic
    MeasurementUnit = 5066068
    MeasurementResolutionIsReadOnly = 0
    MeasurementResolution = 0.01
    CountDirectionIsReadOnly = 0
    CountDirection = Standard
    PeriodSettings:
      Period = 144
  MovementLimitsIsReadOnly = 0
  MovementLimits = Internal
    Position:
      LowerLimitMin = -1.79769313486231E308
      UpperLimitMax = 1.79769313486231E308
      LowerLimit = -1000.0
      UpperLimit = 1000.0
    VelocityIsReadOnly = 0
    Velocity:
      VelocityMax = 3.4E38
      Velocity = 6000
    AccelerationIsReadOnly = 0
    Acceleration:
      AccelerationMax = 3.4E38
      Acceleration = 60000
    DecelerationIsReadOnly = 0
    Deceleration:
      DecelerationMax = 3.4E38
      Deceleration = 60000
  Alarms = MpAlarmX
Element gCutter_MpLink (Type=axis)
  BaseTypeIsReadOnly = 0
  BaseType = RotaryPeriodic
    MeasurementUnitIsReadOnly = 0
    MeasurementUnit = 17476
    MeasurementResolutionIsReadOnly = 0
    MeasurementResolution = 0.01
    CountDirectionIsReadOnly = 0
    CountDirection = Inverse
    PeriodSettings:
      Period = 360
  MovementLimitsIsReadOnly = 0
  MovementLimits = Internal
    Position:
      LowerLimitMin = -1.79769313486231E308
      UpperLimitMax = 1.79769313486231E308
      LowerLimit = -1000.0
      UpperLimit = 1000.0
    VelocityIsReadOnly = 0
    Velocity:
      VelocityMax = 3.4E38
      Velocity = 6000
    AccelerationIsReadOnly = 0
    Acceleration:
      AccelerationMax = 3.4E38
      Acceleration = 60000
    DecelerationIsReadOnly = 0
    Deceleration:
      DecelerationMax = 3.4E38
      Deceleration = 60000
  Alarms = MpAlarmX
```

### Sevos.axis - 5PPC2200_AL14_000/mappMotion/Sevos.axis
```
Element gConv_MpLink (Type=axis)
  BaseTypeIsReadOnly = 0
  BaseType = Linear
    MeasurementUnit = 5066068
    MeasurementResolutionIsReadOnly = 0
    MeasurementResolution = 0.01
    CountDirectionIsReadOnly = 0
    CountDirection = Standard
  MovementLimitsIsReadOnly = 0
  MovementLimits = Internal
    Position:
      LowerLimitMin = -1.79769313486231E308
      UpperLimitMax = 1.79769313486231E308
      LowerLimit = -1000.0
      UpperLimit = 1000.0
    VelocityIsReadOnly = 0
    Velocity:
      VelocityMax = 3.4E38
      Velocity = 6000
    AccelerationIsReadOnly = 0
    Acceleration:
      AccelerationMax = 3.4E38
      Acceleration = 60000
    DecelerationIsReadOnly = 0
    Deceleration:
      DecelerationMax = 3.4E38
      Deceleration = 60000
  Alarms = MpAlarmX
    mapp.AlarmX.Core.Configuration:
      [0]:
        Message = System problem CONV
      [1]:
        Message = Initialization problem CONV
      [2]:
        Message = Parameter problem CONV
      [3]:
        Message = Operation problem CONV
      [9]:
        Message = Network problem CONV
      [10]:
        Message = Encoder problem CONV
      [19]:
        Message = Movement error limit reached CONV
      [20]:
        Message = HW or SW movement limits reached CONV
      [21]:
        Message = Enable input low CONV
Element gCutter_MpLink (Type=axis)
  BaseTypeIsReadOnly = 0
  BaseType = RotaryPeriodic
    MeasurementUnitIsReadOnly = 0
    MeasurementUnit = 17476
    MeasurementResolutionIsReadOnly = 0
    MeasurementResolution = 0.01
    CountDirectionIsReadOnly = 0
    CountDirection = Inverse
    PeriodSettings:
      Period = 360
  MovementLimitsIsReadOnly = 0
  MovementLimits = Internal
    Position:
      LowerLimitMin = -1.79769313486231E308
      UpperLimitMax = 1.79769313486231E308
      LowerLimit = -1000.0
      UpperLimit = 1000.0
    VelocityIsReadOnly = 0
    Velocity:
      VelocityMax = 3.4E38
      Velocity = 6000
    AccelerationIsReadOnly = 0
    Acceleration:
      AccelerationMax = 3.4E38
      Acceleration = 60000
    DecelerationIsReadOnly = 0
    Deceleration:
      DecelerationMax = 3.4E38
      Deceleration = 60000
  Alarms = MpAlarmX
    mapp.AlarmX.Core.Configuration:
      [1]:
        Message = Initialization problem Cutter
      [2]:
        Message = Parameter problem Cutter
      [4]:
        Message = Data access problem Cutter
      [5]:
        Message = Syntax error Cutter
      [9]:
        Message = Network problem Cutter
      [10]:
        Message = Encoder problem Cutter
      [13]:
        Message = Supply problem Cutter
      [19]:
        Message = Movement error limit  Cutter
      [20]:
        Message = HW or SW movement limits reached Cutter
      [21]:
        Message = Enable input   Cutter
```

### unitsOfser.mappmotioncfg - 5PPC2200_AL14_000/mappMotion/unitsOfser.mappmotioncfg
```
Element MappMotionConfiguration (Type=mappmotioncfg)
  Processing:
    ProcessingTaskClass = 1
```

### Config.mprecipecsv - 5PPC2200_AL14_000/mappServices/Config.mprecipecsv
```
Element gRecipeCsv_CFG (Type=mprecipecsv)
  mapp.Recipe.Csv:
    Format:
      DecimalMark = .
  Alarms = MpAlarmX
```

### Config_5.mpalarmxcore - 5PPC2200_AL14_000/mappServices/Config_5.mpalarmxcore
```
Element MpLinkMachinegAlarmXCore (Type=mpalarmxcore)
  mapp.AlarmX.Core.Configuration:
    [0]:
      Name = Alarm2
      Message = {$IAT/ErrorID2}
      Code = 2056
      Severity = 2
      Behavior = DiscreteValueMonitoring
        Monitoring:
          MonitoredPV = ::gErrorID
          TriggerValues:
            [0] = 2
    [1]:
      Name = Alarm3
      Message = {$IAT/ErrorID3}
      Code = 2056
      Behavior = DiscreteValueMonitoring
        Monitoring:
          MonitoredPV = ::gErrorID
          TriggerValues:
            [0] = 3
    [2]:
      Name = Alarm4
      Message = {$IAT/ErrorID4}
      Code = 2056
      Behavior = DiscreteValueMonitoring
        Monitoring:
          MonitoredPV = ::gErrorID
          TriggerValues:
            [0] = 4
    [3]:
      Name = Alarm5
      Message = {$IAT/ErrorID5}
      Code = 2056
      Behavior = DiscreteValueMonitoring
        Monitoring:
          MonitoredPV = ::gErrorID
          TriggerValues:
            [0] = 5
    [4]:
      Name = Alarm6
      Message = {$IAT/ErrorID6}
      Code = 2056
      Severity = 6
      Behavior = DiscreteValueMonitoring
        Monitoring:
          MonitoredPV = ::gErrorID
          TriggerValues:
            [0] = 6
    [5]:
      Name = Alarm7
      Message = {$IAT/ErrorID7}
      Code = 2056
      Behavior = DiscreteValueMonitoring
        Monitoring:
          MonitoredPV = ::gErrorID
          TriggerValues:
            [0] = 7
    [6]:
      Name = Alarm1
      Message = {$IAT/ErrorID1}
      Code = 2056
      Behavior = DiscreteValueMonitoring
        Monitoring:
          MonitoredPV = ::gErrorID
          TriggerValues:
            [0] = 1
```

### Config_6.mpcomunit - 5PPC2200_AL14_000/mappServices/Config_6.mpcomunit
```
Element gGroup (Type=mpcomunit)
  Display:
    Units:
      0:
        DisplayUnits:
          Metric:
            Code = MTL
          Imperial:
            Code = OZI
          ImperialUS:
            Code = OZA
```

## Configuration Config2

CPU 5PPC2200.AL14-000, AutomationRuntime B4.91, Build 4.1.2, Vc V4.72.3

### Hardware
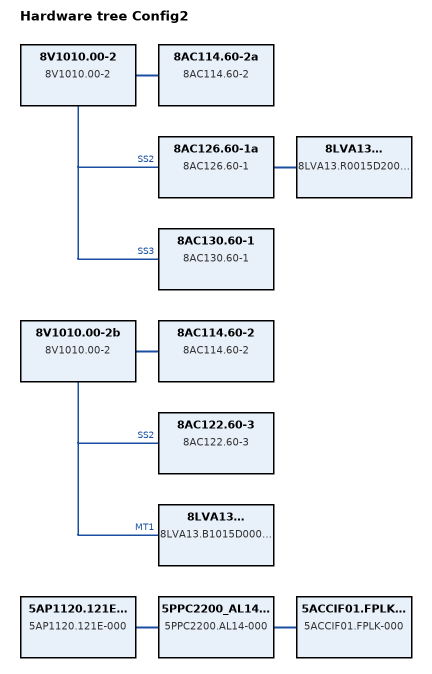
```
5ACCIF01.FPLK-000 : 5ACCIF01.FPLK-000 v1.6.2.0  [SL -> 5PPC2200_AL14_000.SL1]
5AP1120.121E-000 : 5AP1120.121E-000 v2.0.0.0
5PPC2200_AL14_000 : 5PPC2200.AL14-000 v2.0.1.0  [SY -> 5AP1120.121E-000.SY1]
  Connector IF3:
    AssignedOperatingSystem = ARemb
    ActivateDevice = 1
  Connector IF4:
    AssignedOperatingSystem = ARemb
    ActivateDevice = 1
  Connector IF5:
    AssignedOperatingSystem = ARemb
  Connector IF6:
    AssignedOperatingSystem = ARemb
  ConfigurationID = CamAutomat1_Config2
  FileDevice1
  FileDeviceName1 = USER
  FileDevicePath1 = USER_PATH
  ActivateOpcUa = 1
  OpcUaInformationModels_PV_Version = 1
8AC114.60-2 : 8AC114.60-2 v1.0.0.8  [SS -> 8V1010.00-2b.SS1; PLK1 -> 5ACCIF01.FPLK-000.IF1 (NodeNumber=1) [Cable Type=PowerlinkCable, Length=10, Version=1.0.0.3]; PLK2 -> 8AC114.60-2a.PLK1 (NodeNumber=1) [Cable Type=PowerlinkCable, Length=10, Version=1.0.0.3]]
8AC114.60-2a : 8AC114.60-2 v1.0.0.8  [SS -> 8V1010.00-2.SS1; PLK1 -> 8AC114.60-2.PLK2 (NodeNumber=2) [Cable Type=PowerlinkCable, Length=10, Version=1.0.0.3]]
8AC122.60-3 : 8AC122.60-3 v2.2.0.0  [SS -> 8V1010.00-2b.SS2]
  PlugInType = Encoder
  McAcoposTypeID = AcoposPlugInConfig
  ResolverPolepairs = 1
  ResolverTransmissionRatio = 0.5
8AC126.60-1a : 8AC126.60-1 v2.2.0.0  [SS -> 8V1010.00-2.SS2]
  PlugInType = Encoder
  McAcoposTypeID = AcoposPlugInConfig
8AC130.60-1 : 8AC130.60-1 v2.2.0.0  [SS -> 8V1010.00-2.SS3]
8LVA13.B1015D000-0 : 8LVA13.B1015D000-0 v2.2.0.3  [MT -> 8V1010.00-2b.MT1]
  M1/MotorParameters:
    MOTOR_AMB_TEMP_RATED = 40
8LVA13.R0015D200-0 : 8LVA13.R0015D200-0 v2.2.0.3  [EC -> 8AC126.60-1a.EC; MT -> 8V1010.00-2.MT1]
  M1/MotorParameters:
    MOTOR_AMB_TEMP_RATED = 40
8V1010.00-2 : 8V1010.00-2 v2.3.0.0
  DriveConfiguration/Module:
    McAcoposTypeID = AcoposConfig
    ActivateACOPOSSimulationOnPLC = 0
  DriveConfiguration/Channel[1]/RealAxis:
    AxisReference = 
    MechanicalElementsIsInvisible = 0
  DriveConfiguration/Channel[1]/RealAxis/MechanicalElements/Gearbox:
    InputIsReadOnly = 0
    Input = 1
    OutputIsReadOnly = 0
    Output = 1
  DriveConfiguration/Channel[1]/RealAxis/MechanicalElements/RotaryToLinearTransformation:
    ReferenceDistanceIsReadOnly = 0
    ReferenceDistance = 1
  DriveConfiguration/Channel[1]/RealAxis/Controller:
    ModeIsReadOnly = 0
    Mode = PositionController
  DriveConfiguration/Channel[1]/RealAxis/Controller/Mode/Position:
    ProportionalGain = 50.0
    IntegrationTime = 0.0
    PredictionTime = 0.0004
    TotalDelayTime = 0.0004
  DriveConfiguration/Channel[1]/RealAxis/Controller/Mode/Speed:
    ProportionalGainIsReadOnly = 0
    ProportionalGain = 2.0
    IntegrationTimeIsReadOnly = 0
    IntegrationTime = 0.0
    FilterTimeIsReadOnly = 0
    FilterTime = 0.0
  DriveConfiguration/Channel[1]/RealAxis/Controller/Mode/LoopFilters:
    LoopFilterXIsReadOnly = 0
    LoopFilter1 = NotUsed
    LoopFilter2 = NotUsed
    LoopFilter3 = NotUsed
  DriveConfiguration/Channel[1]/RealAxis/Homing:
    ModeIsReadOnly = 0
    Mode = Direct
  DriveConfiguration/Channel[1]/RealAxis/Homing/Mode:
    Position = 0.0
    ReferencePulse = NotUsed
  DriveConfiguration/Channel[1]/RealAxis/Homing:
    RestorePositionVariable = 
  DriveConfiguration/Channel[1]/RealAxis/StopReaction:
    QuickstopIsReadOnly = 0
    Quickstop = DecelerationLimit
    DriveErrorIsReadOnly = 0
    DriveError = DecelerationLimit
  DriveConfiguration/Channel[1]/RealAxis/MovementErrorLimits:
    PositionError = 1.0
    VelocityErrorMonitoring = Automatic1
  DriveConfiguration/Channel[1]/RealAxis:
    JerkFilterIsReadOnly = 0
    JerkFilter = NotUsed
    ZeroVibrationFilter = NotUsed
  DriveConfiguration/Channel[1]/RealAxis/DigitalInputs/HomingSwitch:
    SourceIsReadOnly = 0
    Source = X1Ref
    Level = High
  DriveConfiguration/Channel[1]/RealAxis/DigitalInputs/PositiveLimitSwitch:
    Source = X1PosLim
    Level = High
  DriveConfiguration/Channel[1]/RealAxis/DigitalInputs/NegativeLimitSwitch:
    Source = X1NegLim
    Level = High
  DriveConfiguration/Channel[1]/RealAxis/DigitalInputs/Trigger1:
    Source = X1Trigger1
    Level = High
  DriveConfiguration/Channel[1]/RealAxis/DigitalInputs/Trigger2:
    Source = X1Trigger2
    Level = High
  DriveConfiguration/Channel[1]/RealAxis/DigitalInputs/Quickstop:
    Input = Trigger2
  DriveConfiguration/Channel[1]/RealAxis/Simulation:
    SimulationModeOnPLC = SetValueGeneration
    SimulationModeOnACOPOS = NotUsed
  DriveConfiguration/Channel[1]:
    ExternalEncoderAxis = NotUsed
8V1010.00-2b : 8V1010.00-2 v2.3.0.0
  DriveConfiguration/Module:
    McAcoposTypeID = AcoposConfig
    ActivateACOPOSSimulationOnPLC = 0
  DriveConfiguration/Channel[1]/RealAxis:
    AxisReference = 
    MechanicalElementsIsInvisible = 0
  DriveConfiguration/Channel[1]/RealAxis/MechanicalElements/Gearbox:
    InputIsReadOnly = 0
    Input = 1
    OutputIsReadOnly = 0
    Output = 1
  DriveConfiguration/Channel[1]/RealAxis/MechanicalElements/RotaryToLinearTransformation:
    ReferenceDistanceIsReadOnly = 0
    ReferenceDistance = 1
  DriveConfiguration/Channel[1]/RealAxis/Controller:
    ModeIsReadOnly = 0
    Mode = PositionController
  DriveConfiguration/Channel[1]/RealAxis/Controller/Mode/Position:
    ProportionalGain = 50.0
    IntegrationTime = 0.0
    PredictionTime = 0.0004
    TotalDelayTime = 0.0004
  DriveConfiguration/Channel[1]/RealAxis/Controller/Mode/Speed:
    ProportionalGainIsReadOnly = 0
    ProportionalGain = 2.0
    IntegrationTimeIsReadOnly = 0
    IntegrationTime = 0.0
    FilterTimeIsReadOnly = 0
    FilterTime = 0.0
  DriveConfiguration/Channel[1]/RealAxis/Controller/Mode/LoopFilters:
    LoopFilterXIsReadOnly = 0
    LoopFilter1 = NotUsed
    LoopFilter2 = NotUsed
    LoopFilter3 = NotUsed
  DriveConfiguration/Channel[1]/RealAxis/Homing:
    ModeIsReadOnly = 0
    Mode = Direct
  DriveConfiguration/Channel[1]/RealAxis/Homing/Mode:
    Position = 0.0
    ReferencePulse = NotUsed
  DriveConfiguration/Channel[1]/RealAxis/Homing:
    RestorePositionVariable = 
  DriveConfiguration/Channel[1]/RealAxis/StopReaction:
    QuickstopIsReadOnly = 0
    Quickstop = DecelerationLimit
    DriveErrorIsReadOnly = 0
    DriveError = DecelerationLimit
  DriveConfiguration/Channel[1]/RealAxis/MovementErrorLimits:
    PositionError = 1.0
    VelocityErrorMonitoring = Automatic1
  DriveConfiguration/Channel[1]/RealAxis:
    JerkFilterIsReadOnly = 0
    JerkFilter = NotUsed
    ZeroVibrationFilter = NotUsed
  DriveConfiguration/Channel[1]/RealAxis/DigitalInputs/HomingSwitch:
    SourceIsReadOnly = 0
    Source = X1Ref
    Level = High
  DriveConfiguration/Channel[1]/RealAxis/DigitalInputs/PositiveLimitSwitch:
    Source = X1PosLim
    Level = High
  DriveConfiguration/Channel[1]/RealAxis/DigitalInputs/NegativeLimitSwitch:
    Source = X1NegLim
    Level = High
  DriveConfiguration/Channel[1]/RealAxis/DigitalInputs/Trigger1:
    Source = X1Trigger1
    Level = High
  DriveConfiguration/Channel[1]/RealAxis/DigitalInputs/Trigger2:
    Source = X1Trigger2
    Level = High
  DriveConfiguration/Channel[1]/RealAxis/DigitalInputs/Quickstop:
    Input = Trigger2
  DriveConfiguration/Channel[1]/RealAxis/Simulation:
    SimulationModeOnPLC = SetValueGeneration
    SimulationModeOnACOPOS = NotUsed
  DriveConfiguration/Channel[1]:
    ExternalEncoderAxis = NotUsed
```

## Logical view

Binary libraries used (declarations not repeated): operator, runtime, astime, AsIecCon, brsystem, sys_lib, AsTCP, standard, AsArLog, AsBrStr, MpRecipe, MpBase, McBase, MTTypes, CoTrace, AsZip, FileIO, MpAxis, McAxis, McAcpAx, MpServer, MpAlarmX, MpCom 5.23.1, MTBasics 5.23.0, MpTemp 5.23.0

### Global.typ - Global data types
```iecst
TYPE
	Axis_type : 	STRUCT
		Exists : BOOL;
		name : STRING[10]; (*Name of the axis*)
		cmdReset : BOOL; (*cmd from HMI to reset any fault*)
		cmdStart : BOOL; (*cmd to start this axis *)
		cmdStartAutomat : BOOL;
		cmdCamAutomat : BOOL;
		cmdCam : BOOL;
		cmdGear : BOOL;
		cmdStop : BOOL; (*cmd to stop this axis*)
		cmdHome : BOOL; (*cmd from HMI to home this axis*)
		cmdReference : BOOL; (*cmd from HMI to set the zero offset of the axis.*)
		cmdRun : BOOL; (*cmd to put axis into run state*)
		cmdOffset : BOOL;
		cmdJog : BOOL; (*cmd to put axis into jog state*)
		cmdManualForward : BOOL; (*cmd from HMI to put axis into manual forward state*)
		cmdManualReverse : BOOL; (*cmd from HMI to put axis into manual reverse state*)
		cmdMoveAdditive : BOOL; (*cmd from control task to move axis to absolute position*)
		cmdMoveVelocity : BOOL; (*cmd from control task to move axis to absolute position*)
		cmdMoveAbsolute : BOOL; (*cmd from control task to move axis to absolute position*)
		parmSpeed : REAL; (*cmded speed for manual moves*)
		parmAccelDecel : REAL; (*Acceleration and deceleration of absolute moves*)
		parmAbsolutePosition : REAL; (*Absolute position for absolute moves*)
		parmMaxTorque : REAL; (*Max torque when torque limiting is enabled*)
		statusOn : BOOL; (*Axis is powered on*)
		statusOff : BOOL; (*Axis is powered off*)
		statusDisabled : BOOL; (*Hardware disabled*)
		statusFaulted : BOOL; (*Axis is in the Faulted State*)
		statusStarting : BOOL; (*Axis is in the Starting State*)
		statusHoming : BOOL; (*Axis is in the Homing State*)
		statusInPosition : BOOL; (*Axis is in position following an absolute move*)
		statusRunning : BOOL; (*Axis is in the Running State*)
		statusJogging : BOOL; (*Axis is in the Jogging State*)
		statusMoving : BOOL; (*Axis velocity is > 0*)
		statusManualForward : BOOL; (*Axis is in the Manual Forward State*)
		statusManualReverse : BOOL; (*Axis is in the Manual Reverse State*)
		statusStopping : BOOL; (*Axis is in the Manual Stopping State*)
		statusHomed : BOOL; (*Axis has been homed*)
		statusPosition : LREAL; (*Axis position*)
		statusSpeed : REAL; (*Axis speed*)
		statusCurrent : REAL; (*Axis motor current *)
		statusLagError : REAL; (*Axis lag error*)
		statusTemperature : REAL; (*Actual Temperature*)
		statusTorque : REAL; (*Actual Torque*)
		statusMasterOffset : LREAL; (*Actual offset from master*)
		statusAbsMoveActive : BOOL; (*Absolute move is active*)
		statusGeared : BOOL; (*Axis is geared with the master*)
		statusPoweredOff : BOOL; (*Axis is powered OFF from the software*)
		statusStopped : BOOL; (*Axis has stopped moving*)
		statusPeakCurrent : REAL; (*Peak over the last few seconds motor current *)
		statusPeakLagError : REAL; (*Peak over the last few seconds lag error*)
		statusPeakTorque : REAL; (*Peak over the last few seconds Torque*)
		statusErrorID : UDINT; (*Axis ErrorID (0=no error)*)
		parmMaintMax : REAL;
		parmMaintMin : REAL;
		parmMax : REAL; (*Position to move to when cmded to park. (Real world units)*)
		parmMin : REAL; (*Position to move to when cmded to park. (Real world units)*)
		parmOperMax : REAL; (*Max position displayed on screen based on job setup and mechanical limits*)
		parmOperMin : REAL; (*Min position displayed on screen based on job setup and mechanical limits*)
		parmReferencePosition : REAL; (*Physical position when at the reference mark. (Real world units)*)
	END_STRUCT;
	cutParam_typ : 	STRUCT
		selCutType : UDINT := 1; (*Choose cut type*)
		RecipeName : STRING[65]; (*name of recepit*)
		productionSpeed : REAL := 0.0; (*reference lane *)
		minimumCutSpped : LREAL := 0.0; (*reference lane *)
		lowerPosition : LREAL; (*position Of lower CUT*)
		upperPosition : LREAL; (*position Of Upper CUT*)
	END_STRUCT;
END_TYPE
```

### Global.var - Global variables
```iecst
VAR
	Axis1 : Axis_type := (Exists:=1);
	gCutPosition : LREAL; (*Postition of the conv axis*)
	gConvPosition : LREAL; (*Postition of the conv axis*)
	Axis2 : Axis_type := (Exists:=1); (*Axis 2 setup*)
	CutStart : BOOL; (*User demand cut*)
	Data : ARRAY[0..5] OF LREAL; (*TBD used for Trending too;s*)
	gErrorID : USINT; (*Error ID is used in alarm managment *)
	gReceiptChanged : BOOL; (*Recepit is changed in Hmi need to save date *)
	gSaveParameter : BOOL; (*Paramter is changed in HMI*)
	gServoInitialized : BOOL; (*Initialize servo ad wait for power on*)
	gDispalyServoNotReady : BOOL; (*Not  ready to start  so message will dispal*)
	gEnableTouchProbe : BOOL; (*Enable the touch probe*)
	gCutJogSpeed : REAL := 10.00; (*Jog Speed Cut*)
	gConvPrSpeed : REAL := 3200; (*Product  Speed Conveyor*)
	gConvJogSpeed : REAL := 72.00; (*Jog Speed Conveyor*)
	gManualActive : BOOL; (*Des activate Manaul in the run mode*)
END_VAR
VAR RETAIN
	gMachineStatusArray : ARRAY[0..9] OF STRING[100] := ['Stop/Manual','Run','Manual','Error','Initializing','Finishing Production','PowerOff',3('')]; (*machine status message*)
	gMachineStatusMessage : STRING[100]; (*machine status message array*)
END_VAR
VAR
	gMachineStatus : USINT; (*machine status message*)
END_VAR
VAR RETAIN
	gCutPar : ARRAY[0..2] OF cutParam_typ; (*Recepie parametres*)
END_VAR
VAR
	gMinValue : LREAL := 65.0; (*minum distance*)
END_VAR
VAR RETAIN
	gRecepitRefHmi : INT := 0; (*HMI refrence *)
END_VAR
VAR
	gRunPage : BOOL := FALSE; (*set to on in run from hmi to plc*)
	gResetCount : BOOL; (*Reset number of Count*)
	gvalidDateCamExist : BOOL := FALSE; (*If a Valid Data Exist to trasnfer to cam*)
END_VAR
```

### Package Logical/Libraries - Global libraries

### Library Logical/Libraries/ComTCP/ComTCP_L (ANSIC)

#### MNG_Global.hpp
```cpp
#ifndef  _MNGGLOBAL_HPP_
#define _MNGGLOBAL_HPP_

#include <mng_globalTYP.h>

    typedef struct {

		signed short NumSignals;

        /* BOOL diUnloaded */
        BOOL diUnloaded;
        /* BOOL diLiftUnload */
        BOOL diLiftUnload;
        /* BOOL diLiftTop */
        BOOL diLiftTop;
        /* BOOL diBoxLift */
        BOOL diBoxLift;
        /* BOOL diLiftBottom */
        BOOL diLiftBottom;
        /* BOOL diConvBottom */
        BOOL diConvBottom;
        /* BOOL diConvTop */
        BOOL diConvTop;

        } ComTCP_INPUTS_32BIT_FWRD;

    typedef struct {

		signed short NumSignals;

        /* REAL OutfeedConv_Velocity */
        REAL OutfeedConv_Velocity;
        /* BOOL doLiftTop */
        BOOL doLiftTop;
        /* BOOL doLiftBottom */
        BOOL doLiftBottom;
        /* BOOL doLiftUnload */
        BOOL doLiftUnload;
        /* BOOL doConvLift */
        BOOL doConvLift;
        /* REAL ConvLift_Velocity */
        REAL ConvLift_Velocity;
        /* BOOL doConvBottom */
        BOOL doConvBottom;
        /* REAL ConvBottom_Velocity */
        REAL ConvBottom_Velocity;
        /* LREAL BottomBox_ReleaseTime */
        REAL BottomBox_ReleaseTime;
        /* BOOL doConvTop */
        BOOL doConvTop;
        /* REAL ConvTop_Velocity */
        REAL ConvTop_Velocity;
        /* LREAL TopBox_ReleaseTime */
        REAL TopBox_ReleaseTime;
        /* REAL InfeedConvTop_Velocity */
        REAL InfeedConvTop_Velocity;
        /* REAL InfeedConvBottom_Velocity */
        REAL InfeedConvBottom_Velocity;

        } ComTCP_OUTPUTS_32BIT_FWRD;

#endif
```

#### MNG_CpyMsgToInp.cpp
```cpp
#include "MNG_InternalTyp.hpp"

unsigned long int MNG_CpyMsgToInp(MNG_RawDatagram * pFromServer, ComTCP_INPUTS_32BIT_FWRD *pSimInputs) {

    MNG_DatagramType datagramType;
	unsigned long int DWordBuffer;
        unsigned long int byteCount;
	unsigned long int numSignalsInMessage;

	byteCount = N_TO_HUDINT((pFromServer->Header).ByteCount);
	datagramType = static_cast<MNG_DatagramType>(N_TO_HUDINT((pFromServer->Header).DatagramType));
	if (datagramType != MNG_Raw32BitImage) {
		return 0;
	}

    pSimInputs->NumSignals = 7;

    numSignalsInMessage = N_TO_HUDINT(pFromServer->Payload[0]);
        if ((static_cast<long int>(numSignalsInMessage) != pSimInputs->NumSignals) ||
	(byteCount != 4 + numSignalsInMessage * 4)) {
		return 0;
	}

    /* BOOL diUnloaded */
    pSimInputs->diUnloaded = (pFromServer->Payload[1] != 0);

    /* BOOL diLiftUnload */
    pSimInputs->diLiftUnload = (pFromServer->Payload[2] != 0);

    /* BOOL diLiftTop */
    pSimInputs->diLiftTop = (pFromServer->Payload[3] != 0);

    /* BOOL diBoxLift */
    pSimInputs->diBoxLift = (pFromServer->Payload[4] != 0);

    /* BOOL diLiftBottom */
    pSimInputs->diLiftBottom = (pFromServer->Payload[5] != 0);

    /* BOOL diConvBottom */
    pSimInputs->diConvBottom = (pFromServer->Payload[6] != 0);

    /* BOOL diConvTop */
    pSimInputs->diConvTop = (pFromServer->Payload[7] != 0);

return N_TO_HUDINT((pFromServer->Header).Counter); // return counter
}
```

#### MNG_CpyOutToMsg.cpp
```cpp
#include "MNG_InternalTyp.hpp"

unsigned long int MNG_CpyOutToMsg(MNG_RawDatagram * pToServer, unsigned long int counter, ComTCP_OUTPUTS_32BIT_FWRD *pSimOutputs ) {

        unsigned long int DWordBuffer;

        pSimOutputs->NumSignals = 14;
        (pToServer->Header).ByteCount    = H_TO_NUDINT(60);
        (pToServer->Header).DatagramType = H_TO_NUDINT(MNG_Raw32BitImage);
        (pToServer->Header).SentTime = H_TO_NUDINT(0);  // Todo
        (pToServer->Header).Counter = H_TO_NUDINT(counter);
        pToServer->Payload[0] = H_TO_NUDINT(pSimOutputs->NumSignals);

    /* OutfeedConv_Velocity : FLOAT32 */
    brsmemcpy((unsigned long int)&(DWordBuffer), (unsigned long int)&(pSimOutputs->OutfeedConv_Velocity), 4);
    pToServer->Payload[1] = H_TO_NUDINT(DWordBuffer);

    /* doLiftTop : BOOL */
    if(pSimOutputs->doLiftTop == 1) {
        pToServer->Payload[2] = 0xFFFFFFFF;   /*BOOL */
    } else {
        pToServer->Payload[2] = 0;
    }

    /* doLiftBottom : BOOL */
    if(pSimOutputs->doLiftBottom == 1) {
        pToServer->Payload[3] = 0xFFFFFFFF;   /*BOOL */
    } else {
        pToServer->Payload[3] = 0;
    }

    /* doLiftUnload : BOOL */
    if(pSimOutputs->doLiftUnload == 1) {
        pToServer->Payload[4] = 0xFFFFFFFF;   /*BOOL */
    } else {
        pToServer->Payload[4] = 0;
    }

    /* doConvLift : BOOL */
    if(pSimOutputs->doConvLift == 1) {
        pToServer->Payload[5] = 0xFFFFFFFF;   /*BOOL */
    } else {
        pToServer->Payload[5] = 0;
    }

    /* ConvLift_Velocity : FLOAT32 */
    brsmemcpy((unsigned long int)&(DWordBuffer), (unsigned long int)&(pSimOutputs->ConvLift_Velocity), 4);
    pToServer->Payload[6] = H_TO_NUDINT(DWordBuffer);

    /* doConvBottom : BOOL */
    if(pSimOutputs->doConvBottom == 1) {
        pToServer->Payload[7] = 0xFFFFFFFF;   /*BOOL */
    } else {
        pToServer->Payload[7] = 0;
    }

    /* ConvBottom_Velocity : FLOAT32 */
    brsmemcpy((unsigned long int)&(DWordBuffer), (unsigned long int)&(pSimOutputs->ConvBottom_Velocity), 4);
    pToServer->Payload[8] = H_TO_NUDINT(DWordBuffer);

    /* BottomBox_ReleaseTime : FLOAT64 */
    brsmemcpy((unsigned long int)&(DWordBuffer), (unsigned long int)&(pSimOutputs->BottomBox_ReleaseTime), 4);
    pToServer->Payload[9] = H_TO_NUDINT(DWordBuffer);

    /* doConvTop : BOOL */
    if(pSimOutputs->doConvTop == 1) {
        pToServer->Payload[10] = 0xFFFFFFFF;   /*BOOL */
    } else {
        pToServer->Payload[10] = 0;
    }

    /* ConvTop_Velocity : FLOAT32 */
    brsmemcpy((unsigned long int)&(DWordBuffer), (unsigned long int)&(pSimOutputs->ConvTop_Velocity), 4);
    pToServer->Payload[11] = H_TO_NUDINT(DWordBuffer);

    /* TopBox_ReleaseTime : FLOAT64 */
    brsmemcpy((unsigned long int)&(DWordBuffer), (unsigned long int)&(pSimOutputs->TopBox_ReleaseTime), 4);
    pToServer->Payload[12] = H_TO_NUDINT(DWordBuffer);

    /* InfeedConvTop_Velocity : FLOAT32 */
    brsmemcpy((unsigned long int)&(DWordBuffer), (unsigned long int)&(pSimOutputs->InfeedConvTop_Velocity), 4);
    pToServer->Payload[13] = H_TO_NUDINT(DWordBuffer);

    /* InfeedConvBottom_Velocity : FLOAT32 */
    brsmemcpy((unsigned long int)&(DWordBuffer), (unsigned long int)&(pSimOutputs->InfeedConvBottom_Velocity), 4);
    pToServer->Payload[14] = H_TO_NUDINT(DWordBuffer);

	return 0;
}
```

### MNG_Package.typ
```iecst
(*                                                                            *)
(* File generated by the B&R AS 4 control config generator                    *)
(*                                                                            *)
(*     Provider: machineering                                                 *)
(*  Application: industrialPhysics_2.4.master                                 *)
(* Architecture: Windows 64 Bit                                               *)
(*      Version: 2.4.10898.master                                             *)
(*        Build: 46694f700                                                    *)
(*         Date: 2020-04-28, Time: 08:09:42                                   *)
(*                                                                            *)

TYPE
	ComTCP_INPUTS_32BIT : 	STRUCT
		NumSignals : INT := 7;
		diUnloaded : BOOL := 0; (* BOOL diUnloaded *)
		diLiftUnload : BOOL := 0; (* BOOL diLiftUnload *)
		diLiftTop : BOOL := 0; (* BOOL diLiftTop *)
		diBoxLift : BOOL := 0; (* BOOL diBoxLift *)
		diLiftBottom : BOOL := 0; (* BOOL diLiftBottom *)
		diConvBottom : BOOL := 0; (* BOOL diConvBottom *)
		diConvTop : BOOL := 0; (* BOOL diConvTop *)
	END_STRUCT;
	ComTCP_OUTPUTS_32BIT : 	STRUCT
		NumSignals : INT := 14;
		OutfeedConv_Velocity : REAL := 1; (* REAL OutfeedConv_Velocity *)
		doLiftTop : BOOL := 0; (* BOOL doLiftTop *)
		doLiftBottom : BOOL := 0; (* BOOL doLiftBottom *)
		doLiftUnload : BOOL := 0; (* BOOL doLiftUnload *)
		doConvLift : BOOL := 0; (* BOOL doConvLift *)
		ConvLift_Velocity : REAL := 1; (* REAL ConvLift_Velocity *)
		doConvBottom : BOOL := 0; (* BOOL doConvBottom *)
		ConvBottom_Velocity : REAL := 1; (* REAL ConvBottom_Velocity *)
		BottomBox_ReleaseTime : REAL := 25; (* LREAL BottomBox_ReleaseTime *)
		doConvTop : BOOL := 0; (* BOOL doConvTop *)
		ConvTop_Velocity : REAL := 1; (* REAL ConvTop_Velocity *)
		TopBox_ReleaseTime : REAL := 20; (* LREAL TopBox_ReleaseTime *)
		InfeedConvTop_Velocity : REAL := 0.6; (* REAL InfeedConvTop_Velocity *)
		InfeedConvBottom_Velocity : REAL := 0.5; (* REAL InfeedConvBottom_Velocity *)
	END_STRUCT;
END_TYPE
```

### MNG_Package.var
```iecst
(*                                                                            *)
(* File generated by the B&R AS 4 control config generator                    *)
(*                                                                            *)
(*     Provider: machineering                                                 *)
(*  Application: industrialPhysics_2.4.master                                 *)
(* Architecture: Windows 64 Bit                                               *)
(*      Version: 2.4.10898.master                                             *)
(*        Build: 46694f700                                                    *)
(*         Date: 2020-04-28, Time: 08:09:42                                   *)
(*                                                                            *)
VAR
	ComTCP_SimInputs : ComTCP_INPUTS_32BIT := (0);
	ComTCP_SimOutputs : ComTCP_OUTPUTS_32BIT;
	ComTCP_SimServerAddress : STRING[15] := '127.0.0.1';
	ComTCP_SimServerPort : UINT := 5002;
	ComTCP_SimSendCycleTime : TIME := T#10ms;
	ComTCP_SimActive : BOOL := FALSE;
END_VAR
```

### Package Logical/Images - Imported Images

- Visualisation Logical/mappView (not shown)

### Program Logical/CamAutomat (IEC) - Control Conv. and Cutter

#### Variables.var
```iecst
VAR
	MpAxisBasic_AxisMaster : MpAxisBasic; (*master axis function*)
	AxisParameters_Master : MpAxisBasicParType := (Velocity:=200,Acceleration:=1000,Deceleration:=1000); (*Master paramter defention*)
	MpAxisBasic_AxisSlave : MpAxisBasic; (*master axis function*)
	AxisParameters_Slave : MpAxisBasicParType := (Velocity:=200,Acceleration:=1000,Deceleration:=1000); (*slave axis function paramter *)
	MpAxisCamSequencer_0 : MpAxisCamSequencer; (*cam sequencert*)
	CamSequencerParameters_0 : MpAxisCamSequencerParType; (*cam paramters*)
	Axis2Home : BOOL; (*Home command*)
	Axis1Home : BOOL; (*Home command*)
	Axis1_ErrorID : UINT; (*Error ID Axis 1*)
	AxisStep : UINT; (*Step index for axis*)
	TON_StepDelay : TON := (PT:=T#100ms); (*delay between steps*)
END_VAR
VAR CONSTANT
	STATE_WAIT : USINT := 0; (*State Definition*)
	STATE_POWER_ON : USINT := 1; (*State Definition*)
	STATE_HOME : USINT := 2; (*State Definition*)
	STATE_READY : USINT := 10; (*State Definition*)
	STATE_STOP : USINT := 20; (*State Definition*)
	STATE_MOVE_ABSOLUTE : USINT := 24; (*State Definition*)
	STATE_MOVE_ADDITIVE : USINT := 26; (*State Definition*)
	STATE_MOVE_VELOCITY : USINT := 28; (*State Definition*)
	STATE_MOVE_CAMAUTOMAT : USINT := 30; (*State Definition*)
	STATE_JOG : USINT := 40; (*State Definition*)
	STATE_ERROR : USINT := 101; (*State Definition*)
END_VAR
VAR
	TON_DelayDo1 : TON; (*Timer delay*)
	DelayOpc : TIME := T#20s; (*start up delay*)
	startPositionJog : LREAL; (*potion at where jog start*)
	cutJogEnableBW : BOOL; (*jog backward enable*)
	cutJogEnableFW : BOOL; (*jog reverse enable*)
	bypassProtection : BOOL; (*bypass jog prectoon*)
	displayStopImage : BOOL; (*Display stop image*)
	displayRunImage : BOOL; (*Display Run image*)
	cutEnd : BOOL; (*one cut is done*)
	cutStartDegree : LREAL := 80; (*At this disgree cut start*)
	cutEndDegree : LREAL := 110; (*At this disgree cut end*)
	cutJogEnableFWL : LREAL := 67; (*At this disgree cut jog limit*)
	cutJogEnableFWM : LREAL := 107.5; (*At this disgree cut jog limit*)
	cutJogEnableBWL : LREAL := 71.5; (*At this disgree cut jog limit*)
	sawInCutPosition : BOOL; (*Saw is in cut area*)
	cutJogEnableBWM : LREAL := 112.5; (*At this disgree cut jog limit*)
	displayMessageAuto : BOOL; (*Display message*)
	enableCut : BOOL; (*Enable cut in automatic mode*)
	twoCutEnable : BOOL; (*Enabling two cut from hmi*)
	cutCount : INT; (*Count of Cut*)
	alarmActive : BOOL; (*if there is ana alarm this will be activated*)
	disbaleHome : BOOL; (*disable home in hmi while manual start*)
	maxproducSpeed : REAL; (*maximum probduction Speed*)
	maxSpeed : {REDUND_UNREPLICABLE} REAL := 70.0; (*maximum single cut speed*)
END_VAR
```
